Staubli VAL3: convCreate.pgx

program convCreate(string x_sFileName (dimensions=1), num& x_nError[] (dimensions=1))
  local num l_nError
  local string l_sMessage
  local string l_sSubString
begin
  // This program creates/stores a conveyor library on the flash disk
  //
  // Input Param
  // x_sFileName    : Name of the file for the conveyor library
  //
  // Input Param
  // x_nError      : Error code
  //        0  ->  No Error (success)
  //       35  -> Error while deleting existing conveyor library
  //       36  -> Error while storing new conveyor library
  //       36  -> Error while storing geometry lib
  //
  // Created 23-02-05                                   C.CURRIVAND
  //----------------------------------------------------------------
  //
  x_nError=0
  l_sSubString=cfg:sPATHCONVEYOR+x_sFileName
  call ut:addStrToString(lang:sListOfMessage[34],l_sMessage,"",l_sSubString)
  call up:txtBoxDyn(l_sMessage,3,5,38)
  call up:txtBoxDynUpdate(lang:sListOfMessage[17])
  l_nError=libDelete(cfg:sPATHCONVEYOR+x_sFileName)
  if l_nError==0
    call up:txtBoxDynUpdate(lang:sListOfMessage[18])
    // Setup geometry lib in the conveyor library
    cnv:sGeometryLib=sGeometryLib
    cnv:sConveyorName=x_sFileName
    l_nError=cnv:libSave(cfg:sPATHCONVEYOR+x_sFileName)
    if l_nError==0
      call up:txtBoxDynUpdate(lang:sListOfMessage[19])
      geometry:bIsScara=bIsScara
      call geometry:SetPoint(3)
      l_nError=geometry:libSave(cfg:sPATHCONVEYOR+x_sFileName+"\"+sGeometryLib)
      if l_nError!=0
        // Delete created file(s) if error occured
        libDelete(cfg:sPATHCONVEYOR+x_sFileName)
        // Prepare clear text error message
        x_nError=37
        l_sSubString=cfg:sPATHCONVEYOR+x_sFileName+"\"+sGeometryLib
        call ut:addStrToString(lang:sListOfMessage[x_nError],l_sMessage,"",l_sSubString)
        call ut:addNumToString(l_sMessage,sErrorMessage,"*",l_nError)
      endIf
    else
      // Delete created file(s) if error occured
      libDelete(cfg:sPATHCONVEYOR+x_sFileName)
      // Prepare clear text error message
      x_nError=36
      l_sSubString=cfg:sPATHCONVEYOR+x_sFileName
      call ut:addStrToString(lang:sListOfMessage[x_nError],l_sMessage,"",l_sSubString)
      call ut:addNumToString(l_sMessage,sErrorMessage,"*",l_nError)
    endIf
  else
    // Prepare clear text error message
    x_nError=35
    l_sSubString=cfg:sPATHCONVEYOR+x_sFileName
    call ut:addStrToString(lang:sListOfMessage[x_nError],l_sMessage,"",l_sSubString)
    call ut:addNumToString(l_sMessage,sErrorMessage,"*",l_nError)
  endIf
end
